Fanuc KAREL source: w_d_sys.kl

PROGRAM w_d_sys
%NOLOCKGROUP
%SYSTEM
VAR
  p : POSITION
  r : REAL
BEGIN
  WITH $SPEED = 500 MOVE TO p
  WITH $SPEED = r, $MOTYPE = LINEAR MOVE TO p
END w_d_sys
